Staubli VAL3: remErrCmd.pgx

program remErrCmd(string& sCmd[] (dimensions=1), string& sReturn[] (dimensions=1))
begin
  // Error raised when the command was invalid
  //
  logMsg("call remErrCmd")
  sReturn="ERROR 101"
  sReturn=sReturn+": Invalid command "+sCmd
  putln(sReturn)
  logMsg(sReturn)
end
